FUNCTION_BLOCK PUBLIC FB_File_Write
VAR_INPUT
	bStart  	: REFERENCE TO BOOL;		// Flag operazione
	sFileName 	: REFERENCE TO STRING;		// Nome file + path
	sMess   	: REFERENCE TO STRING;		// messaggio / read / write
	nModeOpen  	: DWORD;					// modalità di apertura
	bOperaz_Ok	: REFERENCE TO BOOL;		// risultato Ok			
	bOperaz_Err : REFERENCE TO BOOL;		// risultato Err
END_VAR
VAR
	// Istanza gestione file 
	fbFileOpen  : FB_FileOpen;		
	fbFileClose : FB_FileClose;
	fbFilePuts  : FB_FilePuts;
	fbFileGets  : FB_FileGets;
	eState 		: (IDLE, OPEN_TRIGGER, OPEN, WRITE_TRIGGER, WRITE, CLOSE_TRIGGER, CLOSE, ERROR, OK );
	bError		: BOOL := FALSE;
END_VAR

IF bStart = TRUE THEN
	eState := OPEN_TRIGGER;
	bStart := FALSE;
	bOperaz_Ok  := FALSE;
	bOperaz_Err := FALSE;
END_IF

CASE eState OF
	IDLE:							// Nulla
	//	
	OPEN_TRIGGER:					// Trigger apertura file
		fbFileOpen(bExecute:=TRUE, sPathName:=sFileName, nMode := nModeOpen);
		eState := OPEN;
	OPEN:							// Attesa file aperto
		fbFileOpen(bExecute:=FALSE);
		IF fbFileOpen.bError THEN
			bError := TRUE;				// -> errore
			eState := ERROR;
		ELSIF NOT fbFileOpen.bBusy AND fbFileOpen.hFile <> 0 THEN
			eState := WRITE_TRIGGER;
		END_IF
	WRITE_TRIGGER:					// Trigger scrittura
		fbFilePuts(bExecute:=TRUE, sLine:=sMess, hFile:=fbFileOpen.hFile );
		eState := WRITE;
	WRITE:							// Attesa scrittura
		fbFilePuts(bExecute:=FALSE);
		IF fbFilePuts.bError THEN
			bError := TRUE;				// -> errore
			eState := CLOSE_TRIGGER;	// -> chiude file
		ELSIF NOT fbFilePuts.bBusy THEN
			eState := CLOSE_TRIGGER;
		END_IF
	CLOSE_TRIGGER:					// Trigger chiusura
		fbFileClose(bExecute:=TRUE, hFile:=fbFileOpen.hFile );
		eState := CLOSE;
	CLOSE:							// Attesa chiusura
		fbFileClose(bExecute:=FALSE);
		IF fbFileClose.bError THEN
			eState := ERROR;
			bError := TRUE;				// -> errore
		ELSIF NOT fbFileClose.bBusy THEN
			IF bError = FALSE THEN
				eState := OK;
			ELSE			
				eState := ERROR;
			END_IF
		END_IF
	OK:								// Fine scrittura Ok
		bOperaz_Ok  := TRUE;
		bOperaz_Err := FALSE;
		eState := IDLE;
	ERROR:							// Fine scrittura Error
		bOperaz_Ok  := FALSE;
		bOperaz_Err := TRUE;
		eState := IDLE;
	
END_CASE

END_FUNCTION_BLOCK

(* stored: Version 1.1.0.1, ProductVersion 3.1.4024.11
   POU FB_File_Write: Id {2ad9d562-e66e-4e0d-a542-ad8e29d25e76}, SpecialFunc None *)
